Fanuc KAREL source: NM0071.KL

-- PROVISIONAL review KL for V1013-1; original PC SHA256 6d0f851da9611bf38a01fdcffa8e829ec1de76eca8bfc37dfdcacb1d3ff76515
-- Incomplete behavior may be omitted. Consult companion uncertainty JSON. Do not deploy.
PROGRAM NM0071
%NOLOCKGROUP
-- UNRESOLVED_LOCAL_POOL 5 cells at code offset 71; source declarations unknown
-- DIRECT_LOCAL_WORD_ACCESS alone does not prove INTEGER, REAL, or BOOLEAN
BEGIN
  -- UNRESOLVED_PC offsets 0-1; opcodes 7B
  -- UNRESOLVED_PC offsets 6-18; opcodes 2D,9D,52,7F
  -- UNRESOLVED_PC offsets 23-28; opcodes 7F,7B
  -- UNRESOLVED_PC offsets 33-49; opcodes 2D,2E,69,7F
  -- UNRESOLVED_PC offsets 54-76; opcodes 7F,2B,2C,7B
  -- UNRESOLVED_PC offsets 81-88; opcodes 9D,23
  -- UNRESOLVED_PC offsets 93-104; opcodes 2E,23
  -- UNRESOLVED_PC offsets 109-120; opcodes 2E,23
  -- UNRESOLVED_PC offsets 125-136; opcodes 2E,23
  -- UNRESOLVED_PC offsets 141-148; opcodes 9D,23
  -- UNRESOLVED_PC offsets 153-162; opcodes 3F,75
  -- UNRESOLVED_PC offsets 167-181; opcodes 2E,22,9D,33,35
  -- UNRESOLVED_PC offsets 186-200; opcodes 2E,22,9D,33,35
  -- UNRESOLVED_PC offsets 205-222; opcodes 27,27,21,64,76,23
  -- UNRESOLVED_PC offsets 227-231; opcodes 7F
  -- UNRESOLVED_PC offsets 236-240; opcodes 27,AA
  -- UNRESOLVED_PC offsets 245-249; opcodes 7F
END NM0071
